PROGRAM MAIN
VAR
	fbDispSens : FB_DisplacementSensor();
END_VAR

END_PROGRAM

(* stored: Version 1.1.0.1, ProductVersion 3.1.4024.12
   POU MAIN: Id {ffa8b730-dc39-431b-9799-d3bf2636dc18}, SpecialFunc None *)
